// SIMATIC S7-200 project (STEP 7-Micro/WIN), CPU 222 REL 01.22

SYMBOL_TABLE USUARIO1
FR1              I0.0     // RELE TERMICO
S1               I0.1     // PULSDOR PARO
S2               I0.2     // PULSADOR MARCHA DERECHA
S3               I0.3     // `PULSADOR MARCHA IZQUIERDAA
KM1              Q0.0     // CONTACTOR MARCHA DERECHA
H1               Q0.1     // SEÑALIZACION MARCHA DERECHA
KM2              Q0.2     // CONTACTOR MARCHA IZQUIERDA
H2               Q0.3     // SEÑALIZACION MARCHA IZQUIERDA
H3               Q0.4     // SEÑALIZACION AVERIA
H4               Q0.5     // SEÑALIZACION PARADA
END_SYMBOL_TABLE

ORGANIZATION_BLOCK PRINCIPAL:OB1
TITLE=COMENTARIOS DEL PROGRAMA
BEGIN
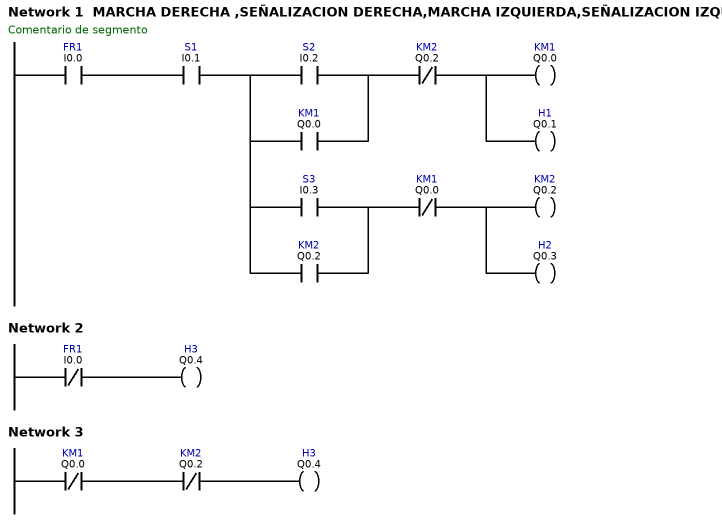
Network 1 // MARCHA DERECHA ,SEÑALIZACION DERECHA,MARCHA IZQUIERDA,SEÑALIZACION IZQUIERDA
.
// Comentario de segmento
// (network saved uncompiled; LAD cells follow)
// row 0: c0 -| |- FR1:I0.0  c1 -| |- S1:I0.1 v  c2 -| |- S2:I0.2 v  c3 -|/|- KM2:Q0.2 v  c4 -( ) KM1:Q0.0
// row 1: c1 ^v  c2 -| |- KM1:Q0.0 ^  c3 ^  c4 -( ) H1:Q0.1
// row 2: c1 ^v  c2 -| |- S3:I0.3 v  c3 -|/|- KM1:Q0.0 v  c4 -( ) KM2:Q0.2
// row 3: c1 ^  c2 -| |- KM2:Q0.2 ^  c3 ^  c4 -( ) H2:Q0.3
Network 2
LDN    FR1:I0.0
=      H3:Q0.4
Network 3
LDN    KM1:Q0.0
AN     KM2:Q0.2
=      H3:Q0.4
END_ORGANIZATION_BLOCK
